// TIA Portal V19 export
TYPE "C103_VAR_IF_OVN_TYPIC"
   STRUCT
      SCL1 { ExternalAccessible := 'False'; ExternalVisible := 'False'; ExternalWritable := 'False'} : Bool;   // Standmelding aankomstschakelaar normaal
      SCL2 { ExternalAccessible := 'False'; ExternalVisible := 'False'; ExternalWritable := 'False'} : Bool;   // Standmelding aankomstschakelaar no-break
      BEV { ExternalAccessible := 'False'; ExternalVisible := 'False'; ExternalWritable := 'False'} : Bool;   // Standmelding automaat kast verwarming en ventilatie
   END_STRUCT;
END_TYPE
